// TIA Portal V17 export
// export: Created 2025-03-07T09:23:42.3674928Z, ExportSetting WithDefaults, DisplayName Totally Integrated Automation Portal, DisplayVersion V17 Update 8, DisplayName TIA Portal Openness, DisplayVersion V17 Update 8, DisplayName TIA Portal Version Control Interface, DisplayVersion V17, DisplayName SINAMICS Startdrive Advanced, DisplayVersion V17 SP2, DisplayName SINAMICS Startdrive G110M, G120, G120C, G120D, G120P, G115D, DisplayVersion V17 SP2, DisplayName SINAMICS Startdrive G130, G150, S120, S150, SINAMICS MV, S210, DisplayVersion V17 SP2, DisplayName STEP 7 Professional, DisplayVersion V17 Update 8, DisplayName SINUMERIK ONE STEP 7 Toolbox, DisplayVersion V17 Update 12, DisplayName SINUMERIK 840D sl STEP 7 Toolbox, DisplayVersion V17 Update 12, DisplayName STEP 7 Safety, DisplayVersion V17 Update 6, DisplayName WinCC Advanced, DisplayVersion V17 Update 8
DATA_BLOCK "DB2141_HOPPER_UNIT_01_IN_OUT"   // DB2141
{ S7_Optimized_Access := 'FALSE'; DB_Accessible_From_OPC_UA := 'FALSE' }
AUTHOR : ETXETAR
VERSION : 1.0
// stored: AutoNumber false, DBAccessibleFromOPCUA false, DBAccessibleFromWebserver true, IsOnlyStoredInLoadMemory false, IsWriteProtectedInAS false
   VAR
      BUTTONS : Struct
         CONTROL_ON : Bool;
         CONTROL_OFF : Bool;
         HOME_POSITION : Bool;
         AUTOMATIC_MODE : Bool;
         SEMIAUTOMATIC_MODE : Bool;
         MANUAL_MODE : Bool;
         START : Bool;
         STOP_END_OF_CYCLE : Bool;
         INMEDIATE_STOP : Bool;
         RESET_FAULTS : Bool;
      END_STRUCT;
      LAMPS : Struct
         CONTROL_ON : Bool;
         CONTROL_OFF : Bool;
         HOME_POSITION : Bool;
         AUTOMATIC_MODE : Bool;
         SEMIAUTOMATIC_MODE : Bool;
         MANUAL_MODE : Bool;
         START : Bool;
         STOP_END_OF_CYCLE : Bool;
         INMEDIATE_STOP : Bool;
         RESET_FAULTS : Bool;
      END_STRUCT;
   END_VAR
BEGIN
END_DATA_BLOCK
